TYPE ST_Ti5CiA402PdoInput :
STRUCT
    nStatusword : UINT;
    nActualPosition : DINT;
    nActualVelocity : DINT;
    nActualTorqueOrCurrent : INT;
    nModeOfOperationDisplay : SINT;
    nErrorCode : UINT;
    nTemperatureRaw : INT;
END_STRUCT
END_TYPE

(* stored: Version 1.1.0.1, ProductVersion 3.1.4024.0 *)
